{attribute addProperty BoxType "EPP3752-0000-0017"}
{attribute addProperty Id "AI_Inputs_ChannelAT %I*ARRAY[0..10] OF AI_Inputs_Channel_83E63207192240WcStateAT %I*WcState_98A4DF7520.250InfoDataAT %I*InfoData_BC63D37F80100"}
{attribute addProperty CRC "3167856318"}
{attribute addProperty SizeInBites "274"}
{attribute addProperty SizeInBytes "34.25"}
TYPE EPP3752_639ED5F3 :
STRUCT
	{attribute addProperty Name "AI_Inputs_Channel"}
	AI_Inputs_Channel : ARRAY[0..10] OF AI_Inputs_Channel_83E63207;
	{attribute addProperty Name "WcState"}
	WcState : WcState_98A4DF75;
	{attribute addProperty Name "InfoData"}
	InfoData : InfoData_BC63D37F;
END_STRUCT
END_TYPE

(* stored: Version 1.2.0.0, ProductVersion 3.1.4024.9
   DUT EPP3752_639ED5F3: Id {6a949d88-8d92-4404-acd7-775bb7e49ecc} *)
